// TIA Portal V21 export
TYPE "Std_Destinazioni"
   STRUCT
      Destinazione : Array[0..25] of "Std_Stazioni";
      Dati : Struct
         DestAttivaPresente : Bool;
         DestSelezionataPresente : Bool;
         AlmenoUnaSorgente : Bool;
      END_STRUCT;
   END_STRUCT;
END_TYPE
